FUNCTION_BLOCK PositionTrigger EXTENDS Objective IMPLEMENTS iObjective
VAR_INPUT

	ThresholdPosition	: LREAL;
	TriggerDirection	: Tc2_MC2.MC_Direction;
	TrackModulo			: LREAL;

END_VAR
VAR_OUTPUT
	MoverPastPosition	: BOOL;
END_VAR
VAR
	someMoverPast		: BOOL;
	whichMover			: INT;
	i					: INT;
	moverLastPos		: ARRAY[0..GVL.NUM_MOVERS-1] OF LREAL;		// Positions of tracked movers from last cycle
	moverLastTurns		: ARRAY[0..GVL.NUM_MOVERS-1] OF DINT;		// Turn count of tracked movers from last cycle
	positiveRolloverDetected: BOOL;
	negativeRolloverDetected: BOOL;
END_VAR


MonitorSuccesses();

ACTION MonitorSuccesses:


someMoverPast		:= FALSE;
whichMover			:= 0;


FOR i := 0 TO GVL.NUM_MOVERS-1 DO	
	IF TrackedMovers[i] <> 0 THEN
		
	
		
	
	
		// Determine if a position rollover occured in the last cycle
		IF TrackedMovers[i]^.AxisReference.NcToPlc.ModuloActTurns > moverLastTurns[i] THEN
			positiveRolloverDetected		:= TRUE;
		ELSIF TrackedMovers[i]^.AxisReference.NcToPlc.ModuloActTurns < moverLastTurns[i] THEN
			negativeRolloverDetected		:= TRUE;
		ELSE
			positiveRolloverDetected		:= FALSE;
			negativeRolloverDetected		:= FALSE;
		END_IF
		// Set value for next cycle
		moverLastTurns[i]	:= TrackedMovers[i]^.AxisReference.NcToPlc.ModuloActTurns;
	
		
		// Can combine with above stanza
		IF positiveRolloverDetected THEN
			moverLastPos[i]		:= moverLastPos[i] - TrackModulo;
		ELSIF negativeRolloverDetected THEN
			moverLastPos[i]		:= moverLastPos[i] + TrackModulo;				
		END_IF
		
		
		
		
		
		
		// Watch for movers crossing the threshold position
		IF TriggerDirection = MC_Positive_Direction THEN
			
			IF moverLastPos[i] < ThresholdPosition AND
				TrackedMovers[i]^.AxisReference.NcToPlc.ModuloActPos >= ThresholdPosition THEN
				// Position trigger event detected
				someMoverPast	:= TRUE;
				whichMover		:= i;
			END_IF
			
		ELSIF TriggerDirection = MC_Negative_Direction THEN
			
			IF moverLastPos[i] > ThresholdPosition AND
				TrackedMovers[i]^.AxisReference.NcToPlc.ModuloActPos <= ThresholdPosition THEN
				// Position trigger event detected
				someMoverPast	:= TRUE;
				whichMover		:= i;
			END_IF		
		
		END_IF

		
		
		moverLastPos[i]			:= TrackedMovers[i]^.AxisReference.NcToPlc.ModuloActPos;
		
		
		
		
	ELSE
		IF TriggerDirection = MC_Negative_Direction THEN
			moverLastPos[i]		:= -1E300;	// very negative value, to prevent false-positive triggers on first cycle
		ELSIF TriggerDirection = MC_Positive_Direction THEN
			moverLastPos[i]		:= 1E300;	// very positive value, to prevent false-positive triggers on first cycle
		END_IF
	END_IF

	
	
	
	
END_FOR




IF someMoverPast THEN
	MoverPastPosition		:= TRUE;
//	CurrentMover			REF= TrackedMovers[whichMover]^;
ELSE
	MoverPastPosition		:= FALSE;
//	CurrentMover			REF= 0;		
END_IF
END_ACTION

END_FUNCTION_BLOCK

(* stored: Version 1.1.0.1, ProductVersion 3.1.4024.9
   POU PositionTrigger: Id {2be242dd-21c3-49cc-ab16-707ac1bbd2e6}, SpecialFunc None
   Folder Methods: Id {f50c0fa9-4833-4154-ba84-add89db4f0c8}
   Folder Properties: Id {7eb93cbf-7ee2-486e-b487-7861ee5391ef}
   Action MonitorSuccesses: Id {e9dd629d-8634-4b16-bccb-b96fc6b6cb24} *)
